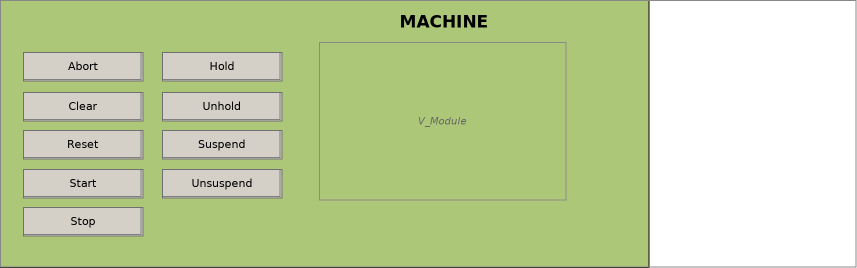
VISUALIZATION V_MachineModule  // 857x268
VAR_IN_OUT
	stVisu				: ST_PMLModuleBaseVISU;
END_VAR
    RoundedRectangle (0,0 649x268)
    Button (23,52 120x29), "Abort"
        tap stVisu.bAbortPressed
    Button (23,92 120x29), "Clear"
        tap stVisu.bClearPressed
    Button (23,130 120x29), "Reset"
        tap stVisu.bResetPressed
    Button (23,169 120x29), "Start"
        tap stVisu.bStartPressed
    Button (23,207 120x29), "Stop"
        tap stVisu.bStopPressed
    Button (162,52 120x29), "Hold"
        tap stVisu.bHoldPressed
    Button (162,92 120x29), "Unhold"
        tap stVisu.bUnholdPressed
    Button (162,130 120x29), "Suspend"
        tap stVisu.bSuspendPressed
    Button (162,169 120x29), "Unsuspend"
        tap stVisu.bUnsuspendPressed
    Frame (319,42 247x158)
        shows V_Module(stVisu := stVisu)
    Label (31,3 826x37), "MACHINE"
END_VISUALIZATION

(* stored: Version 1.1.0.1, ProductVersion 3.1.4024.9
   Visu V_MachineModule: Id {38d3adcf-05a5-497d-bb81-55443dba2d43} *)
